(* CODESYS project tcutilities.library
   Company: TcNexa
   DefaultNamespace: TcNexa_Components_TcUtilities
   Version: 2.0.0
   Placeholder: TcUtilities
   Author: ATI Software Engineering
   Title: TcUtilities

Project tree, tasks and I/O mapping:
  libraries: Tc2_Standard, * (Beckhoff Automation GmbH); Tc2_System, * (Beckhoff Automation GmbH); Tc2_Utilities, * (Beckhoff Automation GmbH); Tc3_Module, * (Beckhoff Automation GmbH); TcProcess, * (TcNexa)
  DUTs/
    data type E_LogSeverity
  String/
    function F_FindAndReplaceAll [ST]
    function F_MemFindString [ST]
    function block FB_ListOfString255 [ST]: _allocateMemory, _deleteMemory, FB_exit, FB_init, size, addToTail, clear, getValueAt
    function block FB_TextSplitter [ST]: size, clear, getValueAt, split
  Tests/
    program PRG_TEST [ST]
  Version/
    global variables Global_Version
  data type T_MaxString
*)

// DUTs/E_LogSeverity
{attribute 'qualified_only'}
{attribute 'strict'}
TYPE E_LogSeverity :
(
	none := 0,
	information,
	warning,
	error
);
END_TYPE

// T_MaxString
TYPE T_MaxString : STRING(255); END_TYPE

// Version/Global_Version
{attribute 'TcGenerated'}
{attribute 'no-analysis'}
{attribute 'linkalways'}
// This function has been automatically generated from the project information.
VAR_GLOBAL CONSTANT
	{attribute 'const_non_replaced'}
	stLibVersion_TcUtilities : ST_LibVersion := (iMajor := 2, iMinor := 0, iBuild := 0, iRevision := 0, nFlags := 0, sVersion := '2.0.0');
END_VAR

// String/F_FindAndReplaceAll
FUNCTION F_FindAndReplaceAll : Tc2_System.T_MaxString
VAR_INPUT
	source			: Tc2_System.T_MaxString;
	toFind			: Tc2_System.T_MaxString;
	toReplaceWith	: Tc2_System.T_MaxString;
END_VAR
VAR
	_value			: UDINT;
END_VAR

_value:= Tc2_Utilities.FindAndReplace(
			pSrcString:= ADR(source),
			pDeleteString:= ADR(toFind),
			pInsertString:= ADR(toReplaceWith),
			pDstString:= ADR(F_FindAndReplaceAll),
			nDstSize:= SIZEOF(F_FindAndReplaceAll));
			
IF (_value = 0) THEN
	F_FindAndReplaceAll:= source;
END_IF

END_FUNCTION

// String/F_MemFindString
(* 0: String not found*)
FUNCTION F_MemFindString : UDINT
VAR_INPUT
	srcAddr			: POINTER TO BYTE;
	toFind			: STRING;
	n				: UDINT;
END_VAR
VAR
	_found			: BOOL;
	_i, _j			: UDINT;
END_VAR

IF (toFind <> '') THEN
	FOR _i:= 0 TO n DO
		IF srcAddr[_i] = toFind[0] THEN
			_found:= TRUE;
			FOR _j:= 0 TO INT_TO_UDINT(Tc2_Standard.LEN(toFind))-1 DO
				IF (srcAddr[_i+_j] <> toFind[_j]) THEN
					_found:= FALSE;
					EXIT;
				END_IF
			END_FOR
			IF _found THEN
				F_MemFindString:= _i+_j;
				EXIT;
			END_IF
		END_IF
	END_FOR
ELSE
	F_MemFindString:= 0;
END_IF

END_FUNCTION

// String/FB_ListOfString255
FUNCTION_BLOCK FB_ListOfString255
VAR
	_list			: POINTER TO Tc2_System.T_MaxString;
	_listSize		: INT;
	_numOfElements	: INT;
	_value			: Tc2_System.T_MaxString;
END_VAR
VAR CONSTANT
	LIST_SIZE		: INT:= 10;
END_VAR

METHOD PROTECTED _allocateMemory : BOOL
VAR_INPUT
END_VAR
VAR
	_tempList			: POINTER TO Tc2_System.T_MaxString;
	_tempListSize		: INT;
END_VAR
_tempListSize:= _listSize + LIST_SIZE;

_tempList:= __NEW(STRING(255), INT_TO_UDINT(_tempListSize));

IF (_listSize > 0) THEN
	Tc2_System.MEMCPY(
		destAddr:= ADR(_tempList[0]), 
		srcAddr	:= ADR(_list[0]), 
		n		:= INT_TO_UDINT(_listSize)*SIZEOF(_value));
	__DELETE(_list);
END_IF

_list:= _tempList;
_listSize:= _tempListSize;
_allocateMemory:= TRUE;
END_METHOD

METHOD PROTECTED _deleteMemory : BOOL
VAR_INPUT
END_VAR
IF (_list <> 0) THEN __DELETE(_list); END_IF
_listSize:= 0;
_numOfElements:= 0;
_deleteMemory:= TRUE;
END_METHOD

METHOD FB_exit : BOOL
VAR_INPUT
	bInCopyCode : BOOL; // if TRUE, the exit method is called for exiting an instance that is copied afterwards (online change).
END_VAR
FB_exit:= NOT bInCopyCode AND_THEN _deleteMemory();
END_METHOD

METHOD FB_init : BOOL
VAR_INPUT
	bInitRetains 	: BOOL; // if TRUE, the retain variables are initialized (warm start / cold start)
	bInCopyCode 	: BOOL;  // if TRUE, the instance afterwards gets moved into the copy code (online change)
END_VAR
IF bInitRetains THEN
	_deleteMemory();
	_allocateMemory();
	FB_init:= TRUE;
END_IF
END_METHOD

PROPERTY PUBLIC size : INT
GET
size:= _numOfElements;
END_GET
END_PROPERTY

METHOD PUBLIC addToTail
VAR_INPUT
	value				: Tc2_System.T_MaxString;
	Response			: REFERENCE TO TcNexa_Components_TcProcess.FB_MethodResponse;
END_VAR
VAR
	_pointer		: POINTER TO Tc2_System.T_MaxString;
END_VAR
IF (_numOfElements >= _listSize) THEN
	_allocateMemory();	
END_IF

_pointer:= (_list + (INT_TO_DWORD(_numOfElements) * SIZEOF(_value)));
IF (_pointer <> 0) THEN
	_pointer^:= value;
	_numOfElements:= _numOfElements + 1;
	IF __ISVALIDREF(Response) THEN Response.setPass(); END_IF
ELSE
	IF __ISVALIDREF(Response) THEN Response.setFail(message:= 'addToTail failed', description:= 'Invalid pointer'); END_IF	
END_IF
END_METHOD

METHOD PUBLIC clear : BOOL
VAR_INPUT
END_VAR
Tc2_System.MEMSET(
	destAddr:= _list,
	fillByte:= 0,
	n		:= INT_TO_UDINT(_numOfElements)*SIZEOF(_value));
_numOfElements:= 0;
clear:= TRUE;
END_METHOD

METHOD PUBLIC getValueAt : Tc2_System.T_MaxString
VAR_INPUT
	index			: INT;
	Response		: REFERENCE TO TcNexa_Components_TcProcess.FB_MethodResponse;
END_VAR
IF (_list = 0) THEN
	IF __ISVALIDREF(Response) THEN Response.setFail(message:= 'getValueAt failed', description:= 'Invalid list address'); END_IF	
ELSIF (_listSize = 0) THEN
	IF __ISVALIDREF(Response) THEN Response.setFail(message:= 'getValueAt failed', description:= 'Invalid list size (size = 0)'); END_IF	
ELSIF (index < 1) THEN
	IF __ISVALIDREF(Response) THEN Response.setFail(message:= 'getValueAt failed', description:= 'Invalid index (index < 1)'); END_IF
ELSIF (index > _listSize) THEN
	IF __ISVALIDREF(Response) THEN Response.setFail(message:= 'getValueAt failed', description:= 'Invalid index (index > list size)'); END_IF
ELSIF (index > _numOfElements) THEN
	IF __ISVALIDREF(Response) THEN Response.setFail(message:= 'getValueAt failed', description:= 'Invalid index (index > number of elements)'); END_IF
ELSE
	getValueAt:= _list[index - 1];	
	IF __ISVALIDREF(Response) THEN Response.setPass(); END_IF					
END_IF
END_METHOD

END_FUNCTION_BLOCK

// String/FB_TextSplitter
FUNCTION_BLOCK FB_TextSplitter
VAR
	_List			: FB_ListOfString255;
END_VAR

PROPERTY PUBLIC size : INT
GET
size:= _List.size;
END_GET
END_PROPERTY

METHOD PUBLIC clear
VAR_INPUT
END_VAR
_List.clear();
END_METHOD

METHOD PUBLIC getValueAt : Tc2_System.T_MaxString
VAR_INPUT
	index		: INT;
	Response	: REFERENCE TO TcNexa_Components_TcProcess.FB_MethodResponse;
END_VAR
getValueAt:= _List.getValueAt(index:= index, Response:= Response);
END_METHOD

METHOD PUBLIC split
VAR_INPUT
	source			: Tc2_System.T_MaxString;
	delimiter		: STRING;
	Response		: REFERENCE TO TcNexa_Components_TcProcess.FB_MethodResponse;
END_VAR
VAR
	_found			: BOOL;
	_leftString		: Tc2_System.T_MaxString;
	_rightString	: Tc2_System.T_MaxString;
END_VAR
clear();

IF (source = '') THEN
	IF __ISVALIDREF(Response) THEN Response.setFail(message:= 'split failed', description:= 'Input string is empty'); END_IF
ELSE
	_rightString:= source;
	
	REPEAT 
		_leftString:= _rightString;
		_found:= Tc2_Utilities.FindAndSplit(
					pSeparator:= ADR(delimiter),
					pSrcString:= ADR(_leftString),
					pLeftString:= ADR(_leftString),
					nLeftSize:= SIZEOF(_leftString),
					pRightString:= ADR(_rightString),
					nRightSize:= SIZEOF(_rightString),
					bSearchFromRight:= FALSE);
					
		_leftString:= F_FindAndReplaceAll(_leftString, '$L', '');
		_leftString:= F_FindAndReplaceAll(_leftString, '$R', '');
		_List.addToTail(value:= _leftString, Response:= 0);
	UNTIL NOT _found
	END_REPEAT
	
	IF __ISVALIDREF(Response) THEN Response.setPass(); END_IF
END_IF
END_METHOD

END_FUNCTION_BLOCK

// Tests/PRG_TEST
PROGRAM PRG_TEST
VAR
END_VAR

END_PROGRAM
